// TwinCAT 3 PLC project gdt_utilities_library
// Title: GDT Utilities Library
// Company: Beckhoff Automation
// Author: GDT
// ProjectVersion: 0.1.0.0
// Description: Graph Development Team utilities library.
// ProgramVersion: 3.1.4023.0
// libraries:
//   Tc2_Standard, * (Beckhoff Automation GmbH)
//   Tc2_System, * (Beckhoff Automation GmbH)
//   Tc2_Utilities, * (Beckhoff Automation GmbH)
//   Tc3_Module, * (Beckhoff Automation GmbH)
//   TcUnit,1.2.0.0,www.tcunit.org
// project tree:
//   DataTypes/FileSystem/ FileExtension.TcDUT, FilePath.TcDUT, FileName.TcDUT
//   / MAIN.TcPOU, PlcTask.TcTTO
//   POUs/FileSystem/- Tests/- Mocks/ Mock_FileSystemEntry.TcPOU
//   POUs/FileSystem/- Tests/ FileEntry_Test.TcPOU, FileSystemEntry_Test.TcPOU, FileSystemEntryCollection_Test.TcPOU, FileSystem_TestSuite.TcPOU, NullEntry_Test.TcPOU, DirectoryEntry_Test.TcPOU
//   POUs/FileSystem/ DirectoryEntry.TcPOU, FileEntry.TcPOU, FileFinder.TcPOU, FileSystemEntry.TcPOU, FileSystemEntryCollection.TcPOU, NullEntry.TcPOU (not stored)
//   POUs/FileSystem/Interfaces/ I_DirectoryEntry.TcIO, I_FileEntry.TcIO, I_FileFinder.TcIO, I_FileSystemEntry.TcIO, I_FileSystemEntryCollection.TcIO, I_NullEntry.TcIO
//   POUs/General/- Tests/ General_TestSuite.TcPOU, IsValueEven_Test.TcPOU, AnyToString_Test.TcPOU, LongStringLen_Test.TcPOU
//   POUs/General/Functions/ AnyToString.TcPOU, IsValueEven.TcPOU, LongStringLen.TcPOU
//   POUs/General/Interfaces/ I_Collection.TcIO, I_Disposable.TcIO (not stored)
//   Version/ Global_Version.TcGVL
// real-time tasks:
//   TASK PlcTask: cycle T#10ms, priority 20, ADS port 350

CONFIGURATION gdt_utilities_library
    RESOURCE PLC ON TwinCAT3
        TASK PlcTask(INTERVAL := T#10ms, PRIORITY := 20);
        PROGRAM MAIN WITH PlcTask : MAIN;
    END_RESOURCE
END_CONFIGURATION

// ---- DataTypes/FileSystem/FileExtension.TcDUT
TYPE FileExtension : STRING(255);
END_TYPE

// ---- DataTypes/FileSystem/FilePath.TcDUT
TYPE FilePath : STRING(255);
END_TYPE

// ---- DataTypes/FileSystem/FileName.TcDUT
TYPE FileName : STRING(255);
END_TYPE

// ---- Version/Global_Version.TcGVL
{attribute 'TcGenerated'}
{attribute 'no-analysis'}
{attribute 'linkalways'}
// This function has been automatically generated from the project information.
VAR_GLOBAL CONSTANT
	{attribute 'const_non_replaced'}
	stLibVersion_GDT_Utilities_Library : ST_LibVersion := (iMajor := 0, iMinor := 1, iBuild := 0, iRevision := 0, nFlags := 0, sVersion := '0.1.0.0');
END_VAR

// ---- POUs/FileSystem/Interfaces/I_DirectoryEntry.TcIO
INTERFACE I_DirectoryEntry EXTENDS I_FileSystemEntry

END_INTERFACE

// ---- POUs/FileSystem/Interfaces/I_FileEntry.TcIO
INTERFACE I_FileEntry EXTENDS I_FileSystemEntry

METHOD GetFullPath : T_MaxString
END_METHOD

PROPERTY Name : FileName
GET
END_GET
SET
END_SET
END_PROPERTY

END_INTERFACE

// ---- POUs/FileSystem/Interfaces/I_FileFinder.TcIO
INTERFACE I_FileFinder EXTENDS __SYSTEM.IQueryInterface

METHOD Find : BOOL;
VAR_INPUT
	SearchDirectory : FilePath;
	FileExtension : FileExtension;
	Collection : I_FileSystemEntryCollection;
END_VAR
END_METHOD

END_INTERFACE

// ---- POUs/FileSystem/Interfaces/I_FileSystemEntry.TcIO
INTERFACE I_FileSystemEntry EXTENDS __SYSTEM.IQueryInterface

PROPERTY PUBLIC IsDirectory : BOOL
GET
END_GET
END_PROPERTY

PROPERTY PUBLIC IsFile : BOOL
GET
END_GET
END_PROPERTY

PROPERTY PUBLIC IsNull : BOOL
GET
END_GET
END_PROPERTY

PROPERTY Path : FilePath
GET
END_GET
END_PROPERTY

END_INTERFACE

// ---- POUs/FileSystem/Interfaces/I_FileSystemEntryCollection.TcIO
INTERFACE I_FileSystemEntryCollection EXTENDS __SYSTEM.IQueryInterface, I_Collection

METHOD Clear
END_METHOD

METHOD GetByIndex : I_FileSystemEntry
VAR_INPUT
	Index : INT;
END_VAR
END_METHOD

METHOD GetFirst : I_FileSystemEntry
END_METHOD

METHOD GetNext : I_FileSystemEntry
VAR_INPUT
	Entry : I_FileSystemEntry;
END_VAR
END_METHOD

METHOD Insert
VAR_INPUT
	Entry : I_FileSystemEntry;
END_VAR
END_METHOD

END_INTERFACE

// ---- POUs/FileSystem/Interfaces/I_NullEntry.TcIO
INTERFACE I_NullEntry EXTENDS I_FileSystemEntry

END_INTERFACE

// ---- POUs/General/Interfaces/I_Collection.TcIO
INTERFACE I_Collection EXTENDS __SYSTEM.IQueryInterface

PROPERTY Count : INT
GET
END_GET
END_PROPERTY

END_INTERFACE

// ---- MAIN.TcPOU
{attribute 'hide'}
PROGRAM MAIN
VAR
	state : (IDLE, FIND_FILES, GET_FILES, DONE) := IDLE;
	
	fileFinder : FileFinder;
	fileCollection : FileSystemEntryCollection;
	searchPath : FilePath := 'C:\temp\integration\';
	fileSystemEntry : I_FileSystemEntry;
	disposable : I_Disposable;
	path : FilePath;
	index : DINT;
END_VAR

General_TestSuite();
FileSystem_TestSuite();

TcUnit.RUN();

// find files in supplied initial folder & sub-folders and populate a collection.
CASE state OF 
	
	IDLE : //
	
	FIND_FILES:
	
		IF (fileFinder.Find(searchPath, '*.tcgraph')) THEN
			state := GET_FILES;
		END_IF
	
	GET_FILES:
		fileCollection := fileFinder.GetResults();	
		fileSystemEntry := fileCollection.GetFirst();
		WHILE NOT (fileSystemEntry.IsNull) DO

			path := fileSystemEntry.Path;
			fileSystemEntry := fileCollection.GetNext(fileSystemEntry);
			
		END_WHILE
		//fileCollection.Clear();
		
		FOR index := 0 TO fileCollection.Count - 1 DO
			fileSystemEntry := fileCollection.GetByIndex(index);
//			IF __QUERYINTERFACE(fileSystemEntry, disposable) THEN
//				disposable.Dispose();
//			END_IF
		END_FOR
		
		state := DONE;
		
	DONE: //
			
	
END_CASE

END_PROGRAM

// ---- POUs/FileSystem/FileFinder.TcPOU
{attribute 'enable_dynamic_creation'}
{attribute 'no_explicit_call' := 'do not call this FB directly'}
FUNCTION_BLOCK PUBLIC FileFinder IMPLEMENTS I_FileFinder, I_Disposable
VAR
	fileCollection : FileSystemEntryCollection;
	status : (INIT, FIRST_READ, NEXT_READ, WAITING_FOR_NOT_BUSY, CHECK_EOE, PROCESS_FOUND_ENTRY, FOUND_DIRECTORY, FOUND_FILE, FINISHED) := INIT;
	searchDir: FilePath;
	searchString : T_MaxString;
	fileExt : FileExtension;
	fbFindFileEntry : FB_EnumFindFileEntry;
	recursiveFileFinder : POINTER TO FileFinder;
END_VAR

METHOD PRIVATE AddNewFileEntryToCollection
VAR_INPUT
	FilePath : FilePath;
	FileEntryData : ST_FindFileEntry;
END_VAR
VAR
	fileEntry : POINTER TO FileEntry;
END_VAR
fileEntry := __NEW(FileEntry(Path:=FilePath, Name:=FileEntryData.sFileName));
THIS^.fileCollection.Insert(fileEntry^);
ADSLOGSTR(ADSLOG_MSGTYPE_STRING, 'File added to collection: %s', fileEntry^.GetFullPath());
END_METHOD

METHOD Dispose
__DELETE(THIS);
END_METHOD

METHOD PRIVATE DisposeEntry
VAR_INPUT
	Entry : I_FileSystemEntry;
END_VAR
VAR
	disposable : I_Disposable;
END_VAR
IF __QUERYINTERFACE(Entry, disposable) THEN
	disposable.Dispose();
END_IF
END_METHOD

METHOD Find : BOOL;
VAR_INPUT
	SearchDirectory : FilePath;
	FileExtension : FileExtension;
END_VAR
VAR
	newSearchDir : FilePath;
	fileEntry : ST_FindFileEntry;
	fileSystemEntry : I_FileSystemEntry;
	recursiveCollection : FileSystemEntryCollection;
END_VAR
CASE status OF
	
	INIT:
		//fileCollection.Clear();
		searchDir := SearchDirectory;
		fileExt := FileExtension;
		searchString := CONCAT(searchDir, '*');
		
		fbFindFileEntry(
			bExecute:=FALSE,
			sNetId:='',
			sPathName:=searchString,
			tTimeout:=DEFAULT_ADS_TIMEOUT
		);
		
		status := FIRST_READ;
		
	FIRST_READ:
		fbFindFileEntry(
			eCmd:=E_EnumCmdType.eEnumCmd_First,
			bExecute:=TRUE,	
		);
		
		status := WAITING_FOR_NOT_BUSY;
	
	NEXT_READ:
		fbFindFileEntry(
			eCmd:=E_EnumCmdType.eEnumCmd_Next,
			bExecute:=TRUE
		);
		
		status := WAITING_FOR_NOT_BUSY;
	
	WAITING_FOR_NOT_BUSY: 
		fbFindFileEntry(bExecute:=FALSE);
		IF NOT fbFindFileEntry.bBusy THEN
			status := CHECK_EOE;
		END_IF

	CHECK_EOE: 
		IF fbFindFileEntry.bEOE THEN
			status := FINISHED;
			RETURN;
		END_IF
		
		status := PROCESS_FOUND_ENTRY;
		
	PROCESS_FOUND_ENTRY:
		IF fbFindFileEntry.stFindFile.fileAttributes.bDirectory THEN
			status := FOUND_DIRECTORY;
			RETURN;
		END_IF
		
		status := FOUND_FILE;
		
	FOUND_DIRECTORY:
	
		IF (fbFindFileEntry.stFindFile.sFileName = '.') OR (fbFindFileEntry.stFindFile.sFileName = '..') THEN
			status := NEXT_READ;
			RETURN;
		END_IF
			
		IF (recursiveFileFinder = 0) THEN				
			recursiveFileFinder := __NEW(FileFinder);
			newSearchDir := CONCAT(searchDir, fbFindFileEntry.stFindFile.sFileName); // sFileName is the name of the directory just found.
			newSearchDir := CONCAT(newSearchDir, '\');
		END_IF

		IF (recursiveFileFinder^.Find(newSearchDir, fileExt)) THEN // find files in sub-directory.
		
			recursiveCollection := recursiveFileFinder^.GetResults();
			fileSystemEntry := recursiveCollection.GetFirst();
		
			WHILE NOT (fileSystemEntry.IsNull) DO
				THIS^.fileCollection.Insert(fileSystemEntry);
				fileSystemEntry := recursiveCollection.GetNext(fileSystemEntry);
			END_WHILE
			
			recursiveCollection.Clear();
			recursiveFileFinder^.Dispose();
			recursiveFileFinder := 0;
			status := NEXT_READ;
			
		END_IF

	FOUND_FILE:
		IF IsMatchingFileExtension(fbFindFileEntry.stFindFile.sFileName, fileExt) THEN
			AddNewFileEntryToCollection(searchDir, fbFindFileEntry.stFindFile);
		END_IF
		
		status := NEXT_READ;
	
	FINISHED:
		Find := TRUE;
		status := INIT;
		RETURN;
	
END_CASE
END_METHOD

METHOD PRIVATE GetFileExtension : FileExtension
VAR_INPUT
	In : FileName;
END_VAR
VAR
	length : INT;
	position : INT;
END_VAR
length := Tc2_Standard.LEN(In);
position := Tc2_Standard.FIND(In, '.');

GetFileExtension := Tc2_Standard.RIGHT(In, (length - position) + 1);
END_METHOD

METHOD GetResults : FileSystemEntryCollection
GetResults := THIS^.fileCollection;
END_METHOD

METHOD PRIVATE IsMatchingFileExtension : BOOL
VAR_INPUT
	In : FileName;
	Extension : FileExtension;
END_VAR
VAR
	extension1 : FileExtension;
	extension2 : FileExtension;
END_VAR
extension1 := GetFileExtension(In);
extension2 := GetFileExtension(Extension);

IsMatchingFileExtension := (extension1 = extension2);
END_METHOD

END_FUNCTION_BLOCK

// ---- POUs/FileSystem/FileSystemEntryCollection.TcPOU
FUNCTION_BLOCK PUBLIC FileSystemEntryCollection IMPLEMENTS I_FileSystemEntryCollection 
VAR
	entries : ARRAY[0..99] OF I_FileSystemEntry;
	currentIndex : DINT := EMPTY;
	_nullEntry : NullEntry(Path:='');
END_VAR
VAR CONSTANT
	EMPTY : DINT :=  -1;
END_VAR

METHOD Clear
VAR
	i : DINT;
END_VAR
FOR i := 0 TO currentIndex DO
	entries[i] := 0;
END_FOR

THIS^.currentIndex := EMPTY;
END_METHOD

PROPERTY Count : UDINT
GET
Count := currentIndex + 1;
END_GET
END_PROPERTY

METHOD GetByIndex : I_FileSystemEntry
VAR_INPUT
	Index : DINT;
END_VAR
IF (Index < 0) THEN
	GetByIndex := _nullEntry;
	RETURN;
END_IF

IF (Index > currentIndex) THEN
	GetByIndex := _nullEntry;
	RETURN;
END_IF

GetByIndex := entries[currentIndex];
END_METHOD

METHOD GetFirst : I_FileSystemEntry
IF NOT (Count > 0) THEN
	GetFirst := _nullEntry;
	RETURN;
END_IF

GetFirst := entries[0];
END_METHOD

METHOD GetNext : I_FileSystemEntry
VAR_INPUT
	Entry : I_FileSystemEntry;
END_VAR
VAR
	i : DINT;
END_VAR
IF Count = 0 THEN
	GetNext := _nullEntry;
	RETURN;
END_IF

IF Entry = 0 THEN
	GetNext := GetFirst();
	RETURN;
END_IF

IF Entry = entries[currentIndex] THEN
	GetNext := _nullEntry;
	RETURN;
END_IF

FOR i := 0 TO currentIndex DO
	IF entries[i] = Entry THEN
		GetNext := entries[i+1];
		RETURN;
	END_IF
END_FOR

GetNext := _nullEntry;
END_METHOD

METHOD Insert
VAR_INPUT
	Entry : I_FileSystemEntry;
END_VAR
IF (currentIndex >= 99) THEN
	RETURN;
END_IF

currentIndex := currentIndex + 1;
entries[currentIndex] := Entry;
END_METHOD

END_FUNCTION_BLOCK

// ---- POUs/FileSystem/FileEntry.TcPOU
{attribute 'enable_dynamic_creation'}
{attribute 'no_explicit_call' := 'do not call this FB directly'}
FUNCTION_BLOCK PUBLIC FileEntry EXTENDS FileSystemEntry IMPLEMENTS I_FileEntry
VAR	
	_name : FileName;
END_VAR

METHOD FB_init : BOOL
VAR_INPUT
	bInitRetains : BOOL; // if TRUE, the retain variables are initialized (warm start / cold start)
	bInCopyCode : BOOL;  // if TRUE, the instance afterwards gets moved into the copy code (online change)
	Path : FilePath;
	Name : FileName;
END_VAR
SUPER^.FB_init(bInitRetains,bInCopyCode,Path);
THIS^._name := Name;
END_METHOD

METHOD GetFullPath : T_MaxString
VAR
	fullPath : T_MaxString;
END_VAR
fullPath := CONCAT(fullPath, Path);
fullPath := CONCAT(fullPath, Name);

GetFullPath := fullPath;
END_METHOD

PROPERTY PUBLIC IsFile : BOOL
GET
IsFile := TRUE;
END_GET
END_PROPERTY

PROPERTY Name : FileName
GET
Name := _name;
END_GET
SET
_name := Name;
END_SET
END_PROPERTY

END_FUNCTION_BLOCK

// ---- POUs/FileSystem/FileSystemEntry.TcPOU
{attribute 'enable_dynamic_creation'}
{attribute 'no_explicit_call' := 'do not call this FB directly'}
FUNCTION_BLOCK PUBLIC ABSTRACT FileSystemEntry IMPLEMENTS I_FileSystemEntry, I_Disposable
VAR
	_path : FilePath;	
END_VAR

METHOD Dispose
__DELETE(THIS);
END_METHOD

METHOD FB_init : BOOL
VAR_INPUT
	bInitRetains : BOOL; // if TRUE, the retain variables are initialized (warm start / cold start)
	bInCopyCode : BOOL;  // if TRUE, the instance afterwards gets moved into the copy code (online change)
	Path : FilePath;
END_VAR
THIS^._path := PathCorrection(Path);
END_METHOD

PROPERTY PUBLIC IsDirectory : BOOL
GET
IsDirectory := FALSE;
END_GET
END_PROPERTY

PROPERTY PUBLIC IsFile : BOOL
GET
IsFile := FALSE;
END_GET
END_PROPERTY

PROPERTY PUBLIC IsNull : BOOL
GET
IsNull := FALSE;
END_GET
END_PROPERTY

PROPERTY Path : FilePath
GET
Path := _path;
END_GET
END_PROPERTY

METHOD PRIVATE PathCorrection : FilePath
VAR_INPUT
	PathToCheck : FilePath;
END_VAR
IF (PathToCheck = '') THEN
	PathCorrection := '.\';
	RETURN;
END_IF

IF (RIGHT(PathToCheck, 1) <> '\') THEN
	PathCorrection := CONCAT(PathToCheck, '\');
	RETURN;
END_IF

PathCorrection := PathToCheck;
END_METHOD

END_FUNCTION_BLOCK

// ---- POUs/General/- Tests/General_TestSuite.TcPOU
{attribute 'hide'}
PROGRAM General_TestSuite
VAR
	anyToStringTest : AnyToString_Test;
	isValueEvenTest : IsValueEven_Test;
	longStringLenTest : LongStringLen_Test;
END_VAR

END_PROGRAM

// ---- POUs/General/- Tests/AnyToString_Test.TcPOU
{attribute 'hide'}
FUNCTION_BLOCK AnyToString_Test EXTENDS TcUnit.FB_TestSuite
VAR
END_VAR

ByteReturnsExpected();
WordReturnsExpected();
DwordReturnsExpected();
LwordReturnsExpected();
//DateAndTimeReturnsExpected();
//DtReturnsExpected();
//DateReturnsExpected();
//TimeOfDayReturnsExpected();
//TodReturnsExpected();
RealReturnsExpected();
LrealReturnsExpected();
UsintReturnsExpected();
UintReturnsExpected();
UdintReturnsExpected();
UlintReturnsExpected();
SintReturnsExpected();
IntReturnsExpected();
DintReturnsExpected();
LintReturnsExpected();
//StringReturnsExpected();
//WstringReturnsExpected();

METHOD ByteReturnsExpected
VAR
	expected : STRING;
	actual : STRING;
	value : BYTE;
END_VAR
TEST('ByteReturnsExpected');

// @TEST-FIXTURE
value := BYTE#16#FF;
expected := '255';

// @TEST-RUN
actual := AnyToString(value);

// @TEST-ASSSERT
AssertEquals_String(Expected := expected, Actual := actual, Message := 'BYTE did return expected');

TEST_FINISHED();
END_METHOD

METHOD DintReturnsExpected
VAR
	expected : STRING;
	actual : STRING;
	value : DINT;
END_VAR
TEST('DintdReturnsExpected');

// @TEST-FIXTURE
value := DINT#16#7FFFFFFF;
expected := '2147483647';

// @TEST-RUN
actual := AnyToString(value);

// @TEST-ASSSERT
AssertEquals_String(Expected := expected, Actual := actual, Message := 'DINT did return expected');

TEST_FINISHED();
END_METHOD

METHOD DwordReturnsExpected
VAR
	expected : STRING;
	actual : STRING;
	value : DWORD;
END_VAR
TEST('DwordReturnsExpected');

// @TEST-FIXTURE
value := DWORD#16#FFFFFFFF;
expected := '4294967295';

// @TEST-RUN
actual := AnyToString(value);

// @TEST-ASSSERT
AssertEquals_String(Expected := expected, Actual := actual, Message := 'DWORD did return expected');

TEST_FINISHED();
END_METHOD

METHOD IntReturnsExpected
VAR
	expected : STRING;
	actual : STRING;
	value : INT;
END_VAR
TEST('IntReturnsExpected');

// @TEST-FIXTURE
value := INT#16#7FFF;
expected := '32767';

// @TEST-RUN
actual := AnyToString(value);

// @TEST-ASSSERT
AssertEquals_String(Expected := expected, Actual := actual, Message := 'INT did return expected');

TEST_FINISHED();
END_METHOD

METHOD LintReturnsExpected
VAR
	expected : STRING;
	actual : STRING;
	value : LINT;
END_VAR
TEST('LintReturnsExpected');

// @TEST-FIXTURE
value := LINT#16#7FFFFFFFFFFFFFFF;
expected := '9223372036854775807';

// @TEST-RUN
actual := AnyToString(value);

// @TEST-ASSSERT
AssertEquals_String(Expected := expected, Actual := actual, Message := 'LINT did return expected');

TEST_FINISHED();
END_METHOD

METHOD LrealReturnsExpected
VAR
	expected : STRING;
	actual : STRING;
	value : LREAL;
END_VAR
TEST('LrealReturnsExpected');

// @TEST-FIXTURE
//TODO TwinCAT crashes when trying to use maximum LREAL value.
//value := LREAL#1.7976931348623158E+308;
//expected := '1.7976931348623158E308';

value := LREAL#3.402823E+38;

//TODO LREAL string returns a lower case 'e' instead of upper case 'E"
expected := '3.402823E38';

// @TEST-RUN
actual := AnyToString(value);

// @TEST-ASSSERT
AssertEquals_String(Expected := expected, Actual := actual, Message := 'LREAL did not return expected');

TEST_FINISHED();
END_METHOD

METHOD LwordReturnsExpected
VAR
	expected : STRING;
	actual : STRING;
	value : LWORD;
END_VAR
TEST('LwordReturnsExpected');

// @TEST-FIXTURE
value := LWORD#16#FFFFFFFFFFFFFFFF;
expected := '18446744073709551615';

// @TEST-RUN
actual := AnyToString(value);

// @TEST-ASSSERT
AssertEquals_String(Expected := expected, Actual := actual, Message := 'LWORD did return expected');

TEST_FINISHED();
END_METHOD

METHOD RealReturnsExpected
VAR
	expected : STRING;
	actual : STRING;
	value : REAL;
END_VAR
TEST('RealReturnsExpected');

// @TEST-FIXTURE
value := REAL#3.402823E+38;
expected := '3.402823E38';

// @TEST-RUN
actual := AnyToString(value);

// @TEST-ASSSERT
AssertEquals_String(Expected := expected, Actual := actual, Message := 'REAL did return expected');

TEST_FINISHED();
END_METHOD

METHOD SintReturnsExpected
VAR
	expected : STRING;
	actual : STRING;
	value : SINT;
END_VAR
TEST('SintReturnsExpected');

// @TEST-FIXTURE
value := SINT#16#7F;
expected := '127';

// @TEST-RUN
actual := AnyToString(value);

// @TEST-ASSSERT
AssertEquals_String(Expected := expected, Actual := actual, Message := 'SINT did return expected');

TEST_FINISHED();
END_METHOD

METHOD UdintReturnsExpected
VAR
	expected : STRING;
	actual : STRING;
	value : UDINT;
END_VAR
TEST('UdintdReturnsExpected');

// @TEST-FIXTURE
value := UDINT#16#FFFFFFFF;
expected := '4294967295';

// @TEST-RUN
actual := AnyToString(value);

// @TEST-ASSSERT
AssertEquals_String(Expected := expected, Actual := actual, Message := 'UDINT did return expected');

TEST_FINISHED();
END_METHOD

METHOD UintReturnsExpected
VAR
	expected : STRING;
	actual : STRING;
	value : UINT;
END_VAR
TEST('UintReturnsExpected');

// @TEST-FIXTURE
value := UINT#16#FFFF;
expected := '65535';

// @TEST-RUN
actual := AnyToString(value);

// @TEST-ASSSERT
AssertEquals_String(Expected := expected, Actual := actual, Message := 'UINT did return expected');

TEST_FINISHED();
END_METHOD

METHOD UlintReturnsExpected
VAR
	expected : STRING;
	actual : STRING;
	value : ULINT;
END_VAR
TEST('UlintReturnsExpected');

// @TEST-FIXTURE
value := ULINT#16#FFFFFFFFFFFFFFFF;
expected := '18446744073709551615';

// @TEST-RUN
actual := AnyToString(value);

// @TEST-ASSSERT
AssertEquals_String(Expected := expected, Actual := actual, Message := 'ULINT did return expected');

TEST_FINISHED();
END_METHOD

METHOD UsintReturnsExpected
VAR
	expected : STRING;
	actual : STRING;
	value : USINT;
END_VAR
TEST('UsintReturnsExpected');

// @TEST-FIXTURE
value := USINT#16#FF;
expected := '255';

// @TEST-RUN
actual := AnyToString(value);

// @TEST-ASSSERT
AssertEquals_String(Expected := expected, Actual := actual, Message := 'USINT did return expected');

TEST_FINISHED();
END_METHOD

METHOD WordReturnsExpected
VAR
	expected : STRING;
	actual : STRING;
	value : WORD;
END_VAR
TEST('WordReturnsExpected');

// @TEST-FIXTURE
value := WORD#16#FFFF;
expected := '65535';

// @TEST-RUN
actual := AnyToString(value);

// @TEST-ASSSERT
AssertEquals_String(Expected := expected, Actual := actual, Message := 'WORD did return expected');

TEST_FINISHED();
END_METHOD

END_FUNCTION_BLOCK

// ---- POUs/General/Functions/AnyToString.TcPOU
FUNCTION AnyToString : STRING
VAR_INPUT
	Value : ANY;
END_VAR
VAR
	pAnyBYTE : POINTER TO BYTE; 
	pAnyWORD : POINTER TO WORD; 
	pAnyDWORD : POINTER TO DWORD; 
	pAnyLWORD : POINTER TO LWORD;
	pAnyDATE_AND_TIME : POINTER TO DATE_AND_TIME; 
	pAnyDT : POINTER TO DT;
	pAnyDATE : POINTER TO DATE; 
	pAnyTIME_OF_DAY : POINTER TO TIME_OF_DAY; 
	pAnyTOD : POINTER TO TOD;
	pAnyREAL : POINTER TO REAL; 
	pAnyLREAL : POINTER TO LREAL;
	pAnyUSINT : POINTER TO USINT; 
	pAnyUINT : POINTER TO UINT;
	pAnyUDINT : POINTER TO UDINT; 
	pAnyULINT : POINTER TO ULINT;
	pAnySINT : POINTER TO SINT; 
	pAnyINT : POINTER TO INT;
	pAnyDINT : POINTER TO DINT; 
	pAnyLINT : POINTER TO LINT;
	pAnySTRING : POINTER TO STRING;
	pAnyWSTRING : POINTER TO WSTRING;
END_VAR

IF (Value.TypeClass = __SYSTEM.TYPE_CLASS.TYPE_BYTE) THEN
    pAnyBYTE := Value.pValue; 
    AnyToString := BYTE_TO_STRING(pAnyBYTE^);
	
ELSIF (Value.TypeClass = __SYSTEM.TYPE_CLASS.TYPE_WORD) THEN
    pAnyWORD := Value.pValue; 
    AnyToString  := WORD_TO_STRING(pAnyWORD^);

ELSIF (Value.TypeClass = __SYSTEM.TYPE_CLASS.TYPE_DWORD) THEN
    pAnyDWORD := Value.pValue; 
    AnyToString  := DWORD_TO_STRING(pAnyDWORD^);
	
ELSIF (Value.TypeClass = __SYSTEM.TYPE_CLASS.TYPE_LWORD) THEN
    pAnyLWORD := Value.pValue; 
    AnyToString  := LWORD_TO_STRING(pAnyLWORD^);
	
ELSIF (Value.TypeClass = __SYSTEM.TYPE_CLASS.TYPE_DATEANDTIME) THEN
    pAnyDATE_AND_TIME := Value.pValue; 
    AnyToString  := DT_TO_STRING(pAnyDATE_AND_TIME^);
	
ELSIF (Value.TypeClass = __SYSTEM.TYPE_CLASS.TYPE_DATE) THEN
    pAnyDATE := Value.pValue; 
    AnyToString  := DATE_TO_STRING(pAnyDATE^);
	
ELSIF (Value.TypeClass = __SYSTEM.TYPE_CLASS.TYPE_TIMEOFDAY) THEN
    pAnyTIME_OF_DAY := Value.pValue; 
    AnyToString  := TOD_TO_STRING(pAnyTIME_OF_DAY^);
	
ELSIF (Value.TypeClass = __SYSTEM.TYPE_CLASS.TYPE_REAL) THEN
    pAnyREAL := Value.pValue; 
    AnyToString  := REAL_TO_STRING(pAnyREAL^);
	
ELSIF (Value.TypeClass = __SYSTEM.TYPE_CLASS.TYPE_LREAL) THEN
    pAnyLREAL := Value.pValue; 
    AnyToString  := F_ToUCase(LREAL_TO_STRING(pAnyLREAL^));
	
ELSIF (Value.TypeClass = __SYSTEM.TYPE_CLASS.TYPE_USINT) THEN
    pAnyUSINT := Value.pValue; 
    AnyToString  := USINT_TO_STRING(pAnyUSINT^);
	
ELSIF (Value.TypeClass = __SYSTEM.TYPE_CLASS.TYPE_UINT) THEN
    pAnyUINT := Value.pValue; 
    AnyToString  := UINT_TO_STRING(pAnyUINT^);
	
ELSIF (Value.TypeClass = __SYSTEM.TYPE_CLASS.TYPE_UDINT) THEN
    pAnyUDINT := Value.pValue; 
    AnyToString  := UDINT_TO_STRING(pAnyUDINT^);
	
ELSIF (Value.TypeClass = __SYSTEM.TYPE_CLASS.TYPE_ULINT) THEN
    pAnyULint := Value.pValue; 
    AnyToString  := ULINT_TO_STRING(pAnyULint^);
	
ELSIF (Value.TypeClass = __SYSTEM.TYPE_CLASS.TYPE_SINT) THEN
    pAnySINT := Value.pValue; 
    AnyToString  := SINT_TO_STRING(pAnySINT^);
	
ELSIF (Value.TypeClass = __SYSTEM.TYPE_CLASS.TYPE_INT) THEN
    pAnyINT := Value.pValue; 
    AnyToString  := INT_TO_STRING(pAnyINT^);
	
ELSIF (Value.TypeClass = __SYSTEM.TYPE_CLASS.TYPE_DINT) THEN
    pAnyDINT := Value.pValue; 
    AnyToString  := DINT_TO_STRING(pAnyDINT^);
	
ELSIF (Value.TypeClass = __SYSTEM.TYPE_CLASS.TYPE_LINT) THEN
    pAnyLINT := Value.pValue; 
    AnyToString  := LINT_TO_STRING(pAnyLINT^);
	
ELSIF (Value.TypeClass = __SYSTEM.TYPE_CLASS.TYPE_STRING) THEN
    pAnySTRING := Value.pValue; 
    AnyToString  := pAnySTRING^;
	
ELSIF (Value.TypeClass = __SYSTEM.TYPE_CLASS.TYPE_WSTRING) THEN
    pAnyWSTRING := Value.pValue; 
    AnyToString  := WSTRING_TO_STRING(pAnyWSTRING^);

END_IF

END_FUNCTION

// ---- POUs/General/- Tests/IsValueEven_Test.TcPOU
{attribute 'hide'}
FUNCTION_BLOCK IsValueEven_Test EXTENDS TcUnit.FB_TestSuite

EvenUSINTReturnsTrue();
EvenUINTReturnsTrue();
EvenUDINTReturnsTrue();
EvenULINTReturnsTrue();
EvenSINTReturnsTrue();
EvenINTReturnsTrue();
EvenDINTReturnsTrue();
EvenLINTReturnsTrue();
OddUSINTReturnsFalse();
OddUINTReturnsFalse();
OddUDINTReturnsFalse();
OddULINTReturnsFalse();
OddSINTReturnsFalse();
OddINTReturnsFalse();
OddDINTReturnsFalse();
OddLINTReturnsFalse();

METHOD EvenDINTReturnsTrue
VAR
	result : BOOL;
	value : DINT;
END_VAR
TEST('EvenDINTReturnsTrue');

// @TEST-FIXTURE
value := DINT#2;

// @TEST-RUN
result := IsValueEven(value);

// @TEST-ASSSERT
AssertTrue(Condition := result,
           Message := 'Even DINT did not return TRUE');

TEST_FINISHED();
END_METHOD

METHOD EvenINTReturnsTrue
VAR
	result : BOOL;
	value : INT;
END_VAR
TEST('EvenINTReturnsTrue');

// @TEST-FIXTURE
value := INT#2;

// @TEST-RUN
result := IsValueEven(value);

// @TEST-ASSSERT
AssertTrue(Condition := result,
           Message := 'Even INT did not return TRUE');

TEST_FINISHED();
END_METHOD

METHOD EvenLINTReturnsTrue
VAR
	result : BOOL;
	value : LINT;
END_VAR
TEST('EvenLINTReturnsTrue');

// @TEST-FIXTURE
value := LINT#2;

// @TEST-RUN
result := IsValueEven(value);

// @TEST-ASSSERT
AssertTrue(Condition := result,
           Message := 'Even LINT did not return TRUE');

TEST_FINISHED();
END_METHOD

METHOD EvenSINTReturnsTrue
VAR
	result : BOOL;
	value : SINT;
END_VAR
TEST('EvenSINTReturnsTrue');

// @TEST-FIXTURE
value := SINT#2;

// @TEST-RUN
result := IsValueEven(value);

// @TEST-ASSSERT
AssertTrue(Condition := result,
           Message := 'Even SINT did not return TRUE');

TEST_FINISHED();
END_METHOD

METHOD EvenUDINTReturnsTrue
VAR
	result : BOOL;
	value : UDINT;
END_VAR
TEST('EvenUDINTReturnsTrue');

// @TEST-FIXTURE
value := UDINT#2;

// @TEST-RUN
result := IsValueEven(value);

// @TEST-ASSSERT
AssertTrue(Condition := result,
           Message := 'Even UDINT did not return TRUE');

TEST_FINISHED();
END_METHOD

METHOD EvenUINTReturnsTrue
VAR
	result : BOOL;
	value : UINT;
END_VAR
TEST('EvenUINTReturnsTrue');

// @TEST-FIXTURE
value := UINT#2;

// @TEST-RUN
result := IsValueEven(value);

// @TEST-ASSSERT
AssertTrue(Condition := result,
           Message := 'Even UINT did not return TRUE');

TEST_FINISHED();
END_METHOD

METHOD EvenULINTReturnsTrue
VAR
	result : BOOL;
	value : ULINT;
END_VAR
TEST('EvenULINTReturnsTrue');

// @TEST-FIXTURE
value := ULINT#2;

// @TEST-RUN
result := IsValueEven(value);

// @TEST-ASSSERT
AssertTrue(Condition := result,
           Message := 'Even ULINT did not return TRUE');

TEST_FINISHED();
END_METHOD

METHOD EvenUSINTReturnsTrue
VAR
	result : BOOL;
	value : USINT;
END_VAR
TEST('EvenUSINTReturnsTrue');

// @TEST-FIXTURE
value := USINT#2;

// @TEST-RUN
result := IsValueEven(value);

// @TEST-ASSSERT
AssertTrue(Condition := result,
           Message := 'Even USINT did not return TRUE');

TEST_FINISHED();
END_METHOD

METHOD OddDINTReturnsFalse
VAR
	result : BOOL;
	value : DINT;
END_VAR
TEST('OddDINTReturnsFalse');

// @TEST-FIXTURE
value := DINT#1;

// @TEST-RUN
result := IsValueEven(value);

// @TEST-ASSSERT
AssertFalse(Condition := result,
           Message := 'Odd DINT did not return FALSE');

TEST_FINISHED();
END_METHOD

METHOD OddINTReturnsFalse
VAR
	result : BOOL;
	value : INT;
END_VAR
TEST('OddINTReturnsFalse');

// @TEST-FIXTURE
value := INT#1;

// @TEST-RUN
result := IsValueEven(value);

// @TEST-ASSSERT
AssertFalse(Condition := result,
           Message := 'Odd INT did not return FALSE');

TEST_FINISHED();
END_METHOD

METHOD OddLINTReturnsFalse
VAR
	result : BOOL;
	value : LINT;
END_VAR
TEST('OddLINTReturnsFalse');

// @TEST-FIXTURE
value := LINT#1;

// @TEST-RUN
result := IsValueEven(value);

// @TEST-ASSSERT
AssertFalse(Condition := result,
           Message := 'Odd LINT did not return FALSE');

TEST_FINISHED();
END_METHOD

METHOD OddSINTReturnsFalse
VAR
	result : BOOL;
	value : SINT;
END_VAR
TEST('OddSINTReturnsFalse');

// @TEST-FIXTURE
value := SINT#1;

// @TEST-RUN
result := IsValueEven(value);

// @TEST-ASSSERT
AssertFalse(Condition := result,
           Message := 'Odd SINT did not return FALSE');

TEST_FINISHED();
END_METHOD

METHOD OddUDINTReturnsFalse
VAR
	result : BOOL;
	value : UDINT;
END_VAR
TEST('OddUDINTReturnsFalse');

// @TEST-FIXTURE
value := UDINT#1;

// @TEST-RUN
result := IsValueEven(value);

// @TEST-ASSSERT
AssertFalse(Condition := result,
           Message := 'Odd UDINT did not return FALSE');

TEST_FINISHED();
END_METHOD

METHOD OddUINTReturnsFalse
VAR
	result : BOOL;
	value : UINT;
END_VAR
TEST('OddUINTReturnsFalse');

// @TEST-FIXTURE
value := UINT#1;

// @TEST-RUN
result := IsValueEven(value);

// @TEST-ASSSERT
AssertFalse(Condition := result,
           Message := 'Odd UINT did not return FALSE');

TEST_FINISHED();
END_METHOD

METHOD OddULINTReturnsFalse
VAR
	result : BOOL;
	value : ULINT;
END_VAR
TEST('OddULINTReturnsFalse');

// @TEST-FIXTURE
value := ULINT#1;

// @TEST-RUN
result := IsValueEven(value);

// @TEST-ASSSERT
AssertFalse(Condition := result,
           Message := 'Odd ULINT did not return FALSE');

TEST_FINISHED();
END_METHOD

METHOD OddUSINTReturnsFalse
VAR
	result : BOOL;
	value : USINT;
END_VAR
TEST('OddUSINTReturnsFalse');

// @TEST-FIXTURE
value := USINT#1;

// @TEST-RUN
result := IsValueEven(value);

// @TEST-ASSSERT
AssertFalse(Condition := result,
           Message := 'Odd USINT did not return FALSE');

TEST_FINISHED();
END_METHOD

END_FUNCTION_BLOCK

// ---- POUs/General/Functions/IsValueEven.TcPOU
FUNCTION IsValueEven : BOOL
VAR_INPUT
	Value : ANY_INT;
END_VAR
VAR
	pAnyUSINT : POINTER TO USINT; 
	pAnyUINT : POINTER TO UINT;
	pAnyUDINT : POINTER TO UDINT; 
	pAnyULINT : POINTER TO ULINT;
	pAnySINT : POINTER TO SINT; 
	pAnyINT : POINTER TO INT;
	pAnyDINT : POINTER TO DINT; 
	pAnyLINT : POINTER TO LINT;
	conversion : ULINT;
END_VAR

IF (Value.TypeClass = __SYSTEM.TYPE_CLASS.TYPE_USINT) THEN
    pAnyUSINT := Value.pValue; 
    conversion  := USINT_TO_ULINT(pAnyUSINT^);
	
ELSIF (Value.TypeClass = __SYSTEM.TYPE_CLASS.TYPE_UINT) THEN
    pAnyUINT := Value.pValue; 
    conversion  := UINT_TO_ULINT(pAnyUINT^);
	
ELSIF (Value.TypeClass = __SYSTEM.TYPE_CLASS.TYPE_UDINT) THEN
    pAnyUDINT := Value.pValue; 
    conversion  := UDINT_TO_ULINT(pAnyUDINT^);
	
ELSIF (Value.TypeClass = __SYSTEM.TYPE_CLASS.TYPE_ULINT) THEN
    pAnyULint := Value.pValue; 
    conversion  := pAnyULint^;
	
ELSIF (Value.TypeClass = __SYSTEM.TYPE_CLASS.TYPE_SINT) THEN
    pAnySINT := Value.pValue; 
    conversion  := SINT_TO_ULINT(pAnySINT^);
	
ELSIF (Value.TypeClass = __SYSTEM.TYPE_CLASS.TYPE_INT) THEN
    pAnyINT := Value.pValue; 
    conversion  := INT_TO_ULINT(pAnyINT^);
	
ELSIF (Value.TypeClass = __SYSTEM.TYPE_CLASS.TYPE_DINT) THEN
    pAnyDINT := Value.pValue; 
    conversion  := DINT_TO_ULINT(pAnyDINT^);
	
ELSIF (Value.TypeClass = __SYSTEM.TYPE_CLASS.TYPE_LINT) THEN
    pAnyLINT := Value.pValue; 
    conversion  := LINT_TO_ULINT(pAnyLINT^);

ELSE
	RETURN;
	
END_IF;

IsValueEven := (conversion MOD 2 ) = 0;

END_FUNCTION

// ---- POUs/General/- Tests/LongStringLen_Test.TcPOU
{attribute 'hide'}
FUNCTION_BLOCK LongStringLen_Test EXTENDS TcUnit.FB_TestSuite

EmptyStringReturnsZero();
LongStringReturnsExpected();
ShortStringReturnsExpected();
T_MaxStringReturns255();

METHOD EmptyStringReturnsZero
VAR
	result : UDINT;
	value : STRING := '';
END_VAR
TEST('EmptyStringReturnsZero');

// @TEST-FIXTURE

// @TEST-RUN
result := LongStringLen(value);

// @TEST-ASSSERT
AssertEquals_UDINT(Expected := UDINT#0, Actual := result,
           Message := 'Empty string did not return zero');
		   

TEST_FINISHED();
END_METHOD

METHOD LongStringReturnsExpected
VAR
	result : UDINT;
	value : STRING(300) := '123456789012345678901234567890123456789012345678901234567890123456789012345678901234567890123456789012345678901234567890123456789012345678901234567890123456789012345678901234567890123456789012345678901234567890123456789012345678901234567890123456789012345678901234567890123456789012345678901234567890';
END_VAR
TEST('LongStringReturnsExpected');

// @TEST-FIXTURE

// @TEST-RUN
result := LongStringLen(value);

// @TEST-ASSSERT
AssertEquals_UDINT(Expected := UDINT#300, Actual := result,
           Message := 'Long string did not return expected');

TEST_FINISHED();
END_METHOD

METHOD ShortStringReturnsExpected
VAR
	result : UDINT;
	value : STRING := '1234567890';
END_VAR
TEST('ShortStringReturnsExpected');

// @TEST-FIXTURE

// @TEST-RUN
result := LongStringLen(value);

// @TEST-ASSSERT
AssertEquals_UDINT(Expected := UDINT#10, Actual := result,
           Message := 'Short string did not return expected');
		   

TEST_FINISHED();
END_METHOD

METHOD T_MaxStringReturns255
VAR
	result : UDINT;
	value : T_MaxString :='123456789012345678901234567890123456789012345678901234567890123456789012345678901234567890123456789012345678901234567890123456789012345678901234567890123456789012345678901234567890123456789012345678901234567890123456789012345678901234567890123456789012345';
END_VAR
TEST('T_MaxStringReturns255');

// @TEST-FIXTURE

// @TEST-RUN
result := LongStringLen(value);

// @TEST-ASSSERT
AssertEquals_UDINT(Expected := UDINT#255, Actual := result,
           Message := 'T_MaxString did not return 255');

TEST_FINISHED();
END_METHOD

END_FUNCTION_BLOCK

// ---- POUs/General/Functions/LongStringLen.TcPOU
FUNCTION LongStringLen : UDINT
VAR_INPUT
	In : ANY_STRING;
END_VAR
VAR
	i : UDINT;
END_VAR

IF NOT In.TypeClass = __SYSTEM.TYPE_CLASS.TYPE_STRING THEN
	RETURN;
END_IF

WHILE (In.pValue[i] <> 0) DO
	i := i+1;
END_WHILE

LongStringLen := i;

END_FUNCTION

// ---- POUs/FileSystem/- Tests/FileSystem_TestSuite.TcPOU
{attribute 'hide'}
PROGRAM FileSystem_TestSuite
VAR
	fileSystemEntryTest : FileSystemEntry_Test;
	nullEntryTest : NullEntry_Test;
	dirEntryTest : DirectoryEntry_Test;
	fileEntryTest : FileEntry_Test;
	fileSystemEntryCollectionTest : FileSystemEntryCollection_Test;
END_VAR

END_PROGRAM

// ---- POUs/FileSystem/- Tests/FileSystemEntry_Test.TcPOU
{attribute 'hide'}
FUNCTION_BLOCK FileSystemEntry_Test EXTENDS TcUnit.FB_TestSuite

EmptyPathReturnsExpected();
SuppliedPathReturnsExpected();
PathAppendsBackslashIfRequired();

METHOD EmptyPathReturnsExpected
VAR
	expected : FilePath;
	actual : FilePath;
	mockFileSystemEntry : Mock_FileSystemEntry('');
END_VAR
TEST('EmptyPathReturnsExpected');

// @TEST-FIXTURE
expected := '.\';

// @TEST-RUN
actual := mockFileSystemEntry.Path;

// @TEST-ASSSERT
AssertEquals_STRING(Expected := expected, Actual := actual, Message := 'Empty path did not return expected');

TEST_FINISHED();
END_METHOD

METHOD PathAppendsBackslashIfRequired
VAR
	expected : FilePath;
	actual : FilePath;
	mockFileSystemEntry : Mock_FileSystemEntry('C:\temp');
END_VAR
TEST('PathAppendsBackslashIfRequired');

// @TEST-FIXTURE
expected := 'C:\temp\';

// @TEST-RUN
actual := mockFileSystemEntry.Path;

// @TEST-ASSSERT
AssertEquals_STRING(Expected := expected, Actual := actual, Message := 'Path did not return expected');

TEST_FINISHED();
END_METHOD

METHOD SuppliedPathReturnsExpected
VAR
	expected : FilePath;
	actual : FilePath;
	mockFileSystemEntry : Mock_FileSystemEntry('C:\TestPath\');
END_VAR
TEST('SuppliedPathReturnsExpected');

// @TEST-FIXTURE
expected := 'C:\TestPath\';

// @TEST-RUN
actual := mockFileSystemEntry.Path;

// @TEST-ASSSERT
AssertEquals_STRING(Expected := expected, Actual := actual, Message := 'Did not return expected path');

TEST_FINISHED();
END_METHOD

END_FUNCTION_BLOCK

// ---- POUs/FileSystem/- Tests/- Mocks/Mock_FileSystemEntry.TcPOU
{attribute 'hide'}
FUNCTION_BLOCK PUBLIC Mock_FileSystemEntry EXTENDS FileSystemEntry

END_FUNCTION_BLOCK

// ---- POUs/FileSystem/- Tests/NullEntry_Test.TcPOU
{attribute 'hide'}
FUNCTION_BLOCK NullEntry_Test EXTENDS TcUnit.FB_TestSuite

IsNullReturnsExpected();

METHOD IsNullReturnsExpected
VAR
	result : BOOL;
	nullEntry : NullEntry('');
END_VAR
TEST('IsNullReturnsExpected');

// @TEST-FIXTURE

// @TEST-RUN
result := nullEntry.IsNull;

// @TEST-ASSSERT
AssertTrue(Condition := result, Message := 'IsNull did not return TRUE');

TEST_FINISHED();
END_METHOD

END_FUNCTION_BLOCK

// ---- POUs/FileSystem/- Tests/DirectoryEntry_Test.TcPOU
{attribute 'hide'}
FUNCTION_BLOCK DirectoryEntry_Test EXTENDS TcUnit.FB_TestSuite

IsDirectoryReturnsExpected();

METHOD IsDirectoryReturnsExpected
VAR
	result : BOOL;
	dirEntry : DirectoryEntry('');
END_VAR
TEST('IsDirectoryReturnsExpected');

// @TEST-FIXTURE

// @TEST-RUN
result := dirEntry.IsDirectory;

// @TEST-ASSSERT
AssertTrue(Condition := result, Message := 'IsDirectory did not return TRUE');

TEST_FINISHED();
END_METHOD

END_FUNCTION_BLOCK

// ---- POUs/FileSystem/DirectoryEntry.TcPOU
{attribute 'enable_dynamic_creation'}
{attribute 'no_explicit_call' := 'do not call this FB directly'}
FUNCTION_BLOCK PUBLIC DirectoryEntry EXTENDS FileSystemEntry IMPLEMENTS I_DirectoryEntry
VAR
END_VAR

PROPERTY PUBLIC IsDirectory : BOOL
GET
IsDirectory := TRUE;
END_GET
END_PROPERTY

END_FUNCTION_BLOCK

// ---- POUs/FileSystem/- Tests/FileEntry_Test.TcPOU
{attribute 'hide'}
FUNCTION_BLOCK FileEntry_Test EXTENDS TcUnit.FB_TestSuite

IsFileReturnsExpected();
NameReturnsExpected();
GetFullPathReturnsExpected();

METHOD GetFullPathReturnsExpected
VAR
	expected : FileName;
	actual : FileName;
	fileEntry : FileEntry('C:\temp', 'test.txt');
END_VAR
TEST('GetFullPathReturnsExpected');

// @TEST-FIXTURE

// @TEST-RUN
expected := 'C:\temp\test.txt';
actual := fileEntry.GetFullPath();

// @TEST-ASSSERT
AssertEquals_STRING(Expected := expected, Actual := actual, Message := 'File GetFullPath did not return expected');

TEST_FINISHED();
END_METHOD

METHOD IsFileReturnsExpected
VAR
	result : BOOL;
	fileEntry : FileEntry('', '');
END_VAR
TEST('IsFileReturnsExpected');

// @TEST-FIXTURE

// @TEST-RUN
result := fileEntry.IsFile;

// @TEST-ASSSERT
AssertTrue(Condition := result, Message := 'IsFile did not return TRUE');

TEST_FINISHED();
END_METHOD

METHOD NameReturnsExpected
VAR
	expected : FileName;
	actual : FileName;
	fileEntry : FileEntry('C:\temp', 'test.txt');
END_VAR
TEST('NameReturnsExpected');

// @TEST-FIXTURE

// @TEST-RUN
expected := 'test.txt';
actual := fileEntry.Name;

// @TEST-ASSSERT
AssertEquals_STRING(Expected := expected, Actual := actual, Message := 'File name did not return expected');

TEST_FINISHED();
END_METHOD

END_FUNCTION_BLOCK

// ---- POUs/FileSystem/- Tests/FileSystemEntryCollection_Test.TcPOU
{attribute 'hide'}
FUNCTION_BLOCK FileSystemEntryCollection_Test EXTENDS TcUnit.FB_TestSuite

CountReturnsZeroAfterClear();
CountReturnsExpectedAfterInsert();
GetFirstReturnsNullIfEmpty();
GetNextReturnsNullIfEmpty();
GetFirstReturnsExpected();
GetNextReturnsExpected();

METHOD CountReturnsExpectedAfterInsert
VAR
	expected : UDINT;
	actual : UDINT;
	mockFileSystemEntry : Mock_FilesystemEntry('');
	collection : FileSystemEntryCollection;
END_VAR
TEST('CountReturnsExpectedAfterInsert');

// @TEST-FIXTURE
expected := 2;

// @TEST-RUN
collection.Insert(mockFileSystemEntry);
collection.Insert(mockFileSystemEntry);
actual := collection.Count;

// @TEST-ASSSERT
AssertEquals_UDINT(Expected := expected, Actual := actual, Message := 'Count did not return expected');

TEST_FINISHED();
END_METHOD

METHOD CountReturnsZeroAfterClear
VAR
	expected : UDINT;
	actual : UDINT;
	collection : FileSystemEntryCollection;
END_VAR
TEST('CountReturnsZeroAfterClear');

// @TEST-FIXTURE
expected := 0;

// @TEST-RUN
collection.Clear();
actual := collection.Count;

// @TEST-ASSSERT
AssertEquals_UDINT(Expected := expected, Actual := actual, Message := 'Count did not return zero');

TEST_FINISHED();
END_METHOD

METHOD GetFirstReturnsExpected
VAR
	collection : FileSystemEntryCollection;
	mockFileSystemEntry : Mock_FilesystemEntry('C:\TestPath\');
	entry : I_FileSystemEntry;
	expected : FilePath;
	actual : FilePath;
END_VAR
TEST('GetFirstReturnsExpected');

// @TEST-FIXTURE
expected := 'C:\TestPath\';

// @TEST-RUN
collection.Insert(mockFileSystemEntry);
entry := collection.GetFirst();

actual := entry.Path;

// @TEST-ASSSERT
AssertEquals_STRING(Expected := expected, Actual := actual, Message := 'Did not return expected');

TEST_FINISHED();
END_METHOD

METHOD GetFirstReturnsNullIfEmpty
VAR
	result : BOOL;
	collection : FileSystemEntryCollection;
	entry : I_FileSystemEntry;
END_VAR
TEST('GetFirstReturnsNullIfEmpty');

// @TEST-FIXTURE

// @TEST-RUN
collection.Clear();
entry := collection.GetFirst();
result := entry.IsNull;

// @TEST-ASSSERT
AssertTrue(Condition := result, Message := 'Did not return a null entry');

TEST_FINISHED();
END_METHOD

METHOD GetNextReturnsExpected
VAR
	collection : FileSystemEntryCollection;
	mockFileSystemEntry1 : Mock_FilesystemEntry('C:\TestPath_1\');
	mockFileSystemEntry2 : Mock_FilesystemEntry('C:\TestPath_2\');
	entry : I_FileSystemEntry;
	expected : FilePath;
	actual : FilePath;
END_VAR
TEST('GetNextReturnsExpected');

// @TEST-FIXTURE
expected := 'C:\TestPath_2\';

// @TEST-RUN
collection.Insert(mockFileSystemEntry1);
collection.Insert(mockFileSystemEntry2);
entry := collection.GetFirst();
entry := collection.GetNext(entry);

actual := entry.Path;

// @TEST-ASSSERT
AssertEquals_STRING(Expected := expected, Actual := actual, Message := 'Did not return expected');

TEST_FINISHED();
END_METHOD

METHOD GetNextReturnsNullIfEmpty
VAR
	result : BOOL;
	collection : FileSystemEntryCollection;
	entry : I_FileSystemEntry;
END_VAR
TEST('GetNextReturnsNullIfEmpty');

// @TEST-FIXTURE

// @TEST-RUN
collection.Clear();
entry := collection.GetNext(0);
result := entry.IsNull;

// @TEST-ASSSERT
AssertTrue(Condition := result, Message := 'Did not return a null entry');

TEST_FINISHED();
END_METHOD

END_FUNCTION_BLOCK
